INTERFACE I_Logger

METHOD PUBLIC M_Log : BOOL
VAR_INPUT
	fbMessage:			FB_Message;
END_VAR
END_METHOD

METHOD M_Reset : BOOL
VAR_INPUT
END_VAR
END_METHOD

END_INTERFACE

(* stored: Version 1.1.0.1
   Itf I_Logger: Id {c8546c00-1964-4def-86cd-48ddf720fa88}
   Method M_Log: Id {70349284-7301-41be-b202-535da7461a8a}
   Method M_Reset: Id {39ef31d6-2654-4e8e-884f-b577042c3611} *)
